Fanuc KAREL source: kt00488.KL

-- PROVISIONAL review KL for V940-1; original PC SHA256 c7bae4e304cebbce41b2a9994391fb2e75b4525371d2444ff8cbd56af0a50c72
-- Incomplete behavior may be omitted. Consult companion uncertainty JSON. Do not deploy.
PROGRAM KT00488
%NOLOCKGROUP
VAR
  OUT : BOOLEAN
-- UNRESOLVED_DECL P1 type=000101
-- UNRESOLVED_DECL P2 type=000199
BEGIN
  -- V9_ZERO_TABLE_METADATA_HINT layout=0001; no indexed target words; source/name/runtime held
  -- UNRESOLVED_PC offsets 5-33; opcodes 49,49,7E,AC,23
  -- UNRESOLVED_PC offsets 38-42; opcodes 7F
END KT00488
